SUBAPPLICATION Uebung_089_AX (* Beispiel für E_R_TRIG, mit Plug and Socket *)
  (* Standard: 61499-2; Description: Copyright (c) 2026 Meisterschulen am Ostbahnhof This program and the accompanying materials are made available under the terms of the Eclipse Public License 2.0 which is available at https://www.eclipse.org/legal/epl-2.0/ SPDX-License-Identifier: EPL-2.0 *)
  (* Version 1.0, 2026-09-10, Franz Höpfinger, Meisterschulen am Ostbahnhof, initial API and implementation and/or initial documentation *)
  PACKAGE Uebungen;
  IMPORT logiBUS::io::DI::logiBUS_DI::Input_I1;
  IMPORT logiBUS::io::DI::logiBUS_DI::Input_I2;
  IMPORT logiBUS::io::DQ::logiBUS_DO::Output_Q1;
  IMPORT logiBUS::io::DQ::logiBUS_DO::Output_Q2;
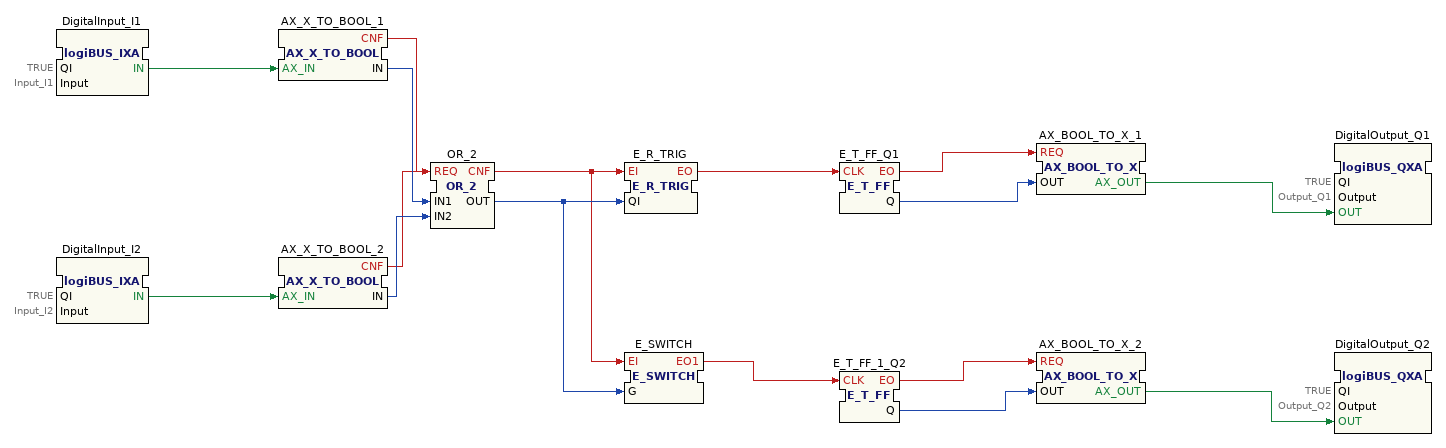
  (* R_TRIG schaltet nur wenn wirklich steigende Flanke *)
  (* E_SWITCH schaltet auch, wenn anderweitig ein Event kommt. *)
  FBS
    DigitalOutput_Q1 : logiBUS::io::DQ::logiBUS_QXA(QI := TRUE, Output := Output_Q1);
    DigitalInput_I1 : logiBUS::io::DI::logiBUS_IXA(QI := TRUE, Input := Input_I1);
    OR_2 : iec61131::bitwiseOperators::OR_2;
    DigitalInput_I2 : logiBUS::io::DI::logiBUS_IXA(QI := TRUE, Input := Input_I2);
    E_R_TRIG : iec61499::events::E_R_TRIG;
    E_T_FF_Q1 : iec61499::events::E_T_FF;
    DigitalOutput_Q2 : logiBUS::io::DQ::logiBUS_QXA(QI := TRUE, Output := Output_Q2);
    E_T_FF_1_Q2 : iec61499::events::E_T_FF;
    E_SWITCH : iec61499::events::E_SWITCH;
    AX_X_TO_BOOL_1 : adapter::conversion::unidirectional::AX_X_TO_BOOL;
    AX_X_TO_BOOL_2 : adapter::conversion::unidirectional::AX_X_TO_BOOL;
    AX_BOOL_TO_X_1 : adapter::conversion::unidirectional::AX_BOOL_TO_X;
    AX_BOOL_TO_X_2 : adapter::conversion::unidirectional::AX_BOOL_TO_X;
  END_FBS
  EVENT_CONNECTIONS
    AX_X_TO_BOOL_2.CNF TO OR_2.REQ;
    AX_X_TO_BOOL_1.CNF TO OR_2.REQ;
    OR_2.CNF TO E_R_TRIG.EI;
    E_R_TRIG.EO TO E_T_FF_Q1.CLK;
    E_T_FF_Q1.EO TO AX_BOOL_TO_X_1.REQ;
    E_SWITCH.EO1 TO E_T_FF_1_Q2.CLK;
    OR_2.CNF TO E_SWITCH.EI;
    E_T_FF_1_Q2.EO TO AX_BOOL_TO_X_2.REQ;
  END_CONNECTIONS
  DATA_CONNECTIONS
    AX_X_TO_BOOL_1.IN TO OR_2.IN1;
    AX_X_TO_BOOL_2.IN TO OR_2.IN2;
    OR_2.OUT TO E_R_TRIG.QI;
    E_T_FF_Q1.Q TO AX_BOOL_TO_X_1.OUT;
    OR_2.OUT TO E_SWITCH.G;
    E_T_FF_1_Q2.Q TO AX_BOOL_TO_X_2.OUT;
  END_CONNECTIONS
  ADAPTER_CONNECTIONS
    DigitalInput_I1.IN TO AX_X_TO_BOOL_1.AX_IN;
    DigitalInput_I2.IN TO AX_X_TO_BOOL_2.AX_IN;
    AX_BOOL_TO_X_1.AX_OUT TO DigitalOutput_Q1.OUT;
    AX_BOOL_TO_X_2.AX_OUT TO DigitalOutput_Q2.OUT;
  END_CONNECTIONS
END_SUBAPPLICATION
